FUNCTION_BLOCK F_LIMIT2 (* limiter *)
  (* Standard: OSCAT *)
  (* Version 0.0, 2011-09-20, 4DIAC-IDE, 4DIAC-Consortium *)
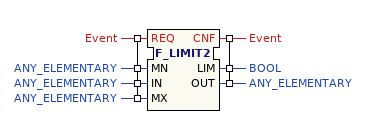
  EVENT_INPUT
    REQ WITH MN, MX, IN; (* Service Request *)
  END_EVENT
  EVENT_OUTPUT
    CNF WITH LIM, OUT; (* Confirmation of Requested Service *)
  END_EVENT
  VAR_INPUT
    MN : ANY_ELEMENTARY; (* Minimum *)
    IN : ANY_ELEMENTARY; (* Input *)
    MX : ANY_ELEMENTARY; (* Maximum *)
  END_VAR
  VAR_OUTPUT
    LIM : BOOL; (* Limit exceeded *)
    OUT : ANY_ELEMENTARY; (* Limited input *)
  END_VAR
  (* Service APPLICATION/RESOURCE: limiter *)
END_FUNCTION_BLOCK
